PROGRAM PRG_Compilation
VAR
	fbHMIManager		: FB_HMIManager;
	fbHMIConfigure		: FB_HMIConfigure;
	
END_VAR

END_PROGRAM

(* stored: Version 1.1.0.1
   POU PRG_Compilation: Id {b568ccfe-ad89-0519-135c-7c4521d3542e}, SpecialFunc None *)
